(* IEC 61131-3 sources: CodesysTest/alpha/export/PackML/OMAC/Function Blocks/UnitModeManager.pou, 5 files *)

(* ---- UnitModeManager.pou.st ---- *)
(*#-#-#-#-#-#-#-#-#-#---Declaration---#-#-#-#-#-#-#-#-#-#-#-#-#*)

// Function block to switch the current unit mode.
{attribute 'hide_all_locals'}
FUNCTION_BLOCK UnitModeManager
VAR_INPUT
END_VAR
VAR_OUTPUT
END_VAR
VAR
	apum: ARRAY[1..gc_usiMaxModes] OF IUnitMode;
	usiNumberOfUMs : USINT := 0;
	usiActualUM: USINT;
END_VAR
(*#-#-#-#-#-#-#-#-#-#---Implementation---#-#-#-#-#-#-#-#-#-#-#-#-#*)

(* ---- AllowsSwitchingTo.m.st ---- *)
(*#-#-#-#-#-#-#-#-#-#---Declaration---#-#-#-#-#-#-#-#-#-#-#-#-#*)

// Checks if the current state allows switching the current unit mode.
{attribute 'hide'}
METHOD PRIVATE AllowsSwitchingTo : BOOL
VAR_INPUT
	usi: USINT; // Unit mode to switch
END_VAR
(*#-#-#-#-#-#-#-#-#-#---Implementation---#-#-#-#-#-#-#-#-#-#-#-#-#*)

IF usi=usiActualUM THEN
	AllowsSwitchingTo := TRUE;
ELSE
	AllowsSwitchingTo := apum[usiActualUM].AllowsLeaving AND apum[usi].AllowsEntering(ActiveUnitMode.CurrentState);
END_IF

(* ---- FindMode.m.st ---- *)
(*#-#-#-#-#-#-#-#-#-#---Declaration---#-#-#-#-#-#-#-#-#-#-#-#-#*)

// Finds an unit mode by name.
{attribute 'hide'}
METHOD PRIVATE FindMode : USINT
VAR_INPUT
	sName: STRING; // Name od the unit mode
END_VAR
VAR
	usi: USINT;
END_VAR(*#-#-#-#-#-#-#-#-#-#---Implementation---#-#-#-#-#-#-#-#-#-#-#-#-#*)

FOR usi := 1 TO usiNumberOfUMs DO
	IF sName = apum[usi].Name THEN
		FindMode := usi;
		RETURN;
	END_IF
END_FOR
FindMode := gc_usiMaxModes+1;

(* ---- Register.m.st ---- *)
(*#-#-#-#-#-#-#-#-#-#---Declaration---#-#-#-#-#-#-#-#-#-#-#-#-#*)

// Registers an unit mode
METHOD Register : BOOL
VAR_INPUT
	pum: IUnitMode;
END_VAR
(*#-#-#-#-#-#-#-#-#-#---Implementation---#-#-#-#-#-#-#-#-#-#-#-#-#*)

IF usiNumberOfUMs < gc_usiMaxModes THEN
	usiNumberOfUMs := usiNumberOfUMs + 1;
	apum[usiNumberOfUMs] := pum;
	IF usiActualUM = 0 THEN
		usiActualUM := 1;
		apum[usiNumberOfUMs].Active := TRUE;
	ELSE
		apum[usiNumberOfUMs].Active := FALSE;
	END_IF
	Register := TRUE;
END_IF

(* ---- SwitchUnitMode.m.st ---- *)
(*#-#-#-#-#-#-#-#-#-#---Declaration---#-#-#-#-#-#-#-#-#-#-#-#-#*)

// Switch to an other unit mode and check the permission.
// Returns true if switching is allowed, returns false if switching is forbidden.
METHOD SwitchUnitMode : BOOL
VAR_INPUT
	sNewModeName: STRING; // Name of the unit mode to switch
END_VAR
VAR
	pnew: POINTER TO UnitMode;
	usi: USINT;
END_VAR(*#-#-#-#-#-#-#-#-#-#---Implementation---#-#-#-#-#-#-#-#-#-#-#-#-#*)

usi := FindMode(sNewModeName);
SwitchUnitMode := FALSE;
IF usi>gc_usiMaxModes THEN
	RETURN;
END_IF

IF usi=usiActualUM THEN
	SwitchUnitMode := TRUE;
	RETURN;
END_IF

IF apum[usiActualUM].AllowsLeaving AND apum[usi].AllowsEntering(ActiveUnitMode.CurrentState) THEN
	apum[usi].Enter(ActiveUnitMode.CurrentState);
	apum[usiActualUM].Active := FALSE;
	apum[usi].Active := TRUE;
	usiActualUM := usi;
	SwitchUnitMode := TRUE;
END_IF
